(* IEC 61131-3 sources: Std_PalletMover/Class/RiwoParamAlarm, 1 file *)

(* ---- RiwoParamAlarm.st ---- *)
(*!
<Class
	Name               = "RiwoParamAlarm"
	Revision           = "0.2"
	RealtimeTask       = "false"
	CyclicTask         = "false"
	BackgroundTask     = "false"
	Sigmatek           = "false"
	OSInterface        = "false"
	HighPriority       = "false"
	Automatic          = "false"
	UpdateMode         = "Prescan"
	SharedCommandTable = "true"
	Objectsize         = "(450,660)">
	<Channels>
		<Server Name="GroupId" Visualized="true" Initialize="true" WriteProtected="false" Retentive="false"/>
		<Server Name="Id" Visualized="true" Initialize="false" WriteProtected="false" Retentive="false"/>
		<Server Name="Level" Visualized="true" Initialize="false" WriteProtected="false" Retentive="SRam"/>
		<Server Name="Parameter1" Visualized="false" Initialize="false" WriteProtected="false" Retentive="false"/>
		<Server Name="Parameter2" Visualized="false" Initialize="false" WriteProtected="false" Retentive="false"/>
		<Server Name="Parameter3" Visualized="false" Initialize="false" WriteProtected="false" Retentive="false"/>
		<Server Name="Parameter4" Visualized="false" Initialize="false" WriteProtected="false" Retentive="false"/>
		<Server Name="Report" Visualized="true" Initialize="false" WriteProtected="false" Retentive="SRam"/>
		<Server Name="ResetReq" Visualized="false" Initialize="true" WriteProtected="false" Retentive="false"/>
		<Client Name="_Group" Required="true" Internal="true"/>
		<Client Name="_Id" Required="true" Internal="true"/>
		<Client Name="objNextRiwoParamAlarm" Required="false" Internal="false"/>
		<Client Name="objRiwoEventLogger" Required="false" Internal="false"/>
	</Channels>
	<Dependencies>
		<Files>
			<File Path=".\Class\RiwoDefine\RiwoDef.h" Include="false"/>
		</Files>
	</Dependencies>
	<RevDoku>
		<Owner Company="Riwo Engineering B.V." Author="Stefan Veltmaat (SVE)"/>
		<Dokumentation Revision="0.1" Date="2018-07-27" Author="Stefan Veltmaat (SVE)" Company="Riwo Engineering B.V." Description="initial setup of parmeter error"/>
		<Dokumentation Date="2018-07-27" Author="Stefan Veltmaat (SVE)" Company="Riwo Engineering B.V."/>
	</RevDoku>
	<Network Name="RiwoParamAlarm">
		<!-- List of Components in this network -->
		<Components>
			<Object
				Name       = "_base"
				Class      = "_AlarmX3Para"
				Position   = "(534,120)"
				Visualized = "true"
				Remotely   = "true">
				<Channels>
					<Server Name="ClassSvr"/>
					<Client Name="Acknow"/>
					<Client Name="Config" Value="0"/>
					<Client Name="Group"/>
					<Client Name="Para1"/>
					<Client Name="Para2"/>
					<Client Name="Para3"/>
				</Channels>
			</Object>
			<Object
				Name       = "_Group"
				Class      = "Ram"
				Position   = "(390,690)"
				Visualized = "true"
				Remotely   = "true">
				<Channels>
					<Server Name="Data"/>
				</Channels>
			</Object>
			<Object
				Name       = "_Id"
				Class      = "Ram"
				Position   = "(390,480)"
				Visualized = "true"
				Remotely   = "true">
				<Channels>
					<Server Name="Data"/>
				</Channels>
			</Object>
		</Components>
		<Comments>
		</Comments>
		<!-- List of Connections in this network -->
		<Connections>
			<Connection Source="this.ClassSvr" Destination="_base.ClassSvr" Vertices="(1006,210),(834,210),"/>
			<Connection Source="this._Group" Destination="_Group.Data"/>
			<Connection Source="this.Id" Destination="_Id.Data" Vertices="(1006,270),(690,570),"/>
			<Connection Source="this.GroupId" Destination="_Group.Data" Vertices="(1006,330),(690,780),"/>
			<Connection Source="this._Id" Destination="_Id.Data"/>
		</Connections>
		<!-- Headerfiles -->
		<Options>
		</Options>
	</Network>
</Class>
*)
#pragma using _AlarmX3Para

RiwoParamAlarm : CLASS
: _AlarmX3Para
	TYPE
	  eAlarmLevel :  //! <Type Public="true" Name="eAlarmLevel"/>
	  (
	    eal_Error,
	    eal_Warning,
	    eal_Info
	  )$UDINT;
	  eAlarmReport :  //! <Type Public="true" Name="eAlarmReport"/>
	  (
	    ear_No,
	    ear_Yes
	  )$UDINT;
	END_TYPE
  //Servers:
	Id 	: SvrCh_DINT;
	GroupId 	: SvrCh_DINT;
	ResetReq 	: SvrCh_DINT;
	Level 	: SvrCh_eAlarmLevel_PTofCls_RiwoParamAlarm;
	Report 	: SvrCh_DINT;
	Parameter1 	: SvrCh_DINT;
	Parameter2 	: SvrCh_DINT;
	Parameter3 	: SvrCh_DINT;
	Parameter4 	: SvrCh_DINT;
  //Clients:
	objRiwoEventLogger 	: CltChCmd_RiwoEventLogger;
	objNextRiwoParamAlarm 	: CltChCmd_RiwoParamAlarm;
	_Id 	: CltChCmd_Ram;
	_Group 	: CltChCmd_Ram;
  //Variables:
  //Functions:

	FUNCTION VIRTUAL GLOBAL Init;

	FUNCTION VIRTUAL GLOBAL GetParaVal
		VAR_INPUT
			ppara 	: ^DINT;
		END_VAR
		VAR_OUTPUT
			retcode 	: UDINT;
		END_VAR;

	FUNCTION VIRTUAL GLOBAL QuitAlarm;

	FUNCTION _HandleAlarms
		VAR_INPUT
			newState 	: DINT;
		END_VAR;

	FUNCTION GLOBAL SetActive;

	FUNCTION GLOBAL SetInActive;

	FUNCTION GLOBAL SetActiveSingleParamAlarm
		VAR_INPUT
			inparam1 	: DINT;
		END_VAR;

	FUNCTION GLOBAL SetActiveTwoParamsAlarm
		VAR_INPUT
			inparam1 	: DINT;
			inparam2 	: DINT;
		END_VAR;

	FUNCTION GLOBAL SetActiveThreeParamsAlarm
		VAR_INPUT
			inparam1 	: DINT;
			inparam2 	: DINT;
			inparam3 	: DINT;
		END_VAR;

	FUNCTION GLOBAL GetActiveErrors
		VAR_INPUT
			objNr 	: UDINT;
		END_VAR
		VAR_OUTPUT
			errorsState 	: BDINT;
		END_VAR;

	FUNCTION GLOBAL GetActiveWarnings
		VAR_INPUT
			objNr 	: UDINT;
		END_VAR
		VAR_OUTPUT
			warningsState 	: BDINT;
		END_VAR;

	FUNCTION GLOBAL GetReportConfigs
		VAR_INPUT
			objNr 	: UDINT;
		END_VAR
		VAR_OUTPUT
			reportConfigs 	: BDINT;
		END_VAR;

	FUNCTION GLOBAL SetAlarmIds
		VAR_INPUT
			startId 	: DINT;
		END_VAR;

	FUNCTION VIRTUAL GLOBAL Id::Read
		VAR_OUTPUT
			output (EAX) 	: DINT;
		END_VAR;

	FUNCTION VIRTUAL GLOBAL Id::Write
		VAR_INPUT
			input (EAX) 	: DINT;
		END_VAR
		VAR_OUTPUT
			result (EAX) 	: DINT;
		END_VAR;

	FUNCTION VIRTUAL GLOBAL GroupId::Read
		VAR_OUTPUT
			output (EAX) 	: DINT;
		END_VAR;

	FUNCTION VIRTUAL GLOBAL GroupId::Write
		VAR_INPUT
			input (EAX) 	: DINT;
		END_VAR
		VAR_OUTPUT
			result (EAX) 	: DINT;
		END_VAR;

	FUNCTION VIRTUAL GLOBAL ResetReq::Read
		VAR_OUTPUT
			output (EAX) 	: DINT;
		END_VAR;

	FUNCTION VIRTUAL GLOBAL ResetReq::Write
		VAR_INPUT
			input (EAX) 	: DINT;
		END_VAR
		VAR_OUTPUT
			result (EAX) 	: DINT;
		END_VAR;
  //Tables:
	FUNCTION @STD
		VAR_OUTPUT
			ret_code	: CONFSTATES;
		END_VAR;
	FUNCTION GLOBAL TAB @CT_;
END_CLASS;

#pragma using Ram
#pragma usingLtd RiwoEventLogger

FUNCTION VIRTUAL GLOBAL RiwoParamAlarm::Init
  #if MAX_ALARMPARA >= 5
    #define ALARMPARA_NR_SUITABLE 1
  #endif

  #pragma warning(disable: 69);
  // compile error look into AlarmXBuffer.h and set MAX_ALARMPARA to 5
  if ALARMPARA_NR_SUITABLE then
    _AlarmX0Para::Init();
  end_if;
  #pragma warning(default: 69);

END_FUNCTION

FUNCTION GLOBAL RiwoParamAlarm::SetActive
  _HandleAlarms(1);
END_FUNCTION

FUNCTION GLOBAL RiwoParamAlarm::SetInActive
  _HandleAlarms(0);
END_FUNCTION

FUNCTION RiwoParamAlarm::_HandleAlarms
	VAR_INPUT
		newState 	: DINT;
	END_VAR

  if Level = eal_Warning & newState <> ClassSvr & newState = 1 then
    _RIWO_WARNING_MSG0("Alarm Id {0} activated", to_dint(Id));

    //write the new state to the ClassSvr so it is handled correct
    ClassSvr.Write(input:= newState);
  elsif Level = eal_Error  & newState <> ClassSvr & newState = 1 then
    _RIWO_ERROR_MSG0("Alarm Id {0} activated", to_dint(Id));

    //write the new state to the ClassSvr so it is handled correct
    ClassSvr.Write(input:= newState);
  elsif newState <> ClassSvr then
    _RIWO_INFO_MSG0("Alarm Id {0} de-activated", to_dint(Id));

    //write the new state to the ClassSvr so it is handled correct
    ClassSvr.Write(input:= newState);
  end_if;

  //all error updates must result in disabling the Reset request signal
  ResetReq := 0;

END_FUNCTION

FUNCTION VIRTUAL GLOBAL RiwoParamAlarm::GetParaVal
	VAR_INPUT
		ppara 	: ^DINT;
	END_VAR
	VAR_OUTPUT
		retcode 	: UDINT;
	END_VAR

  //Param position 0 contains level and report now, first 8 bits are Level, second 8 bits are report.
  ppara^ := Level$DINT AND 255;
  ppara^ := ppara^ OR Report$DINT SHL 8;

  //catch acces exception when sigmatek define is set back to its default of 3 instead of the needed 5
  //otherwise we are writing outside memory

  #if MAX_ALARMPARA >= 5
    ppara += 4;
    ppara^ := Parameter1;
    ppara += 4;
    ppara^ := Parameter2;
    ppara += 4;
    ppara^ := Parameter3;
    ppara += 4;
    ppara^ := Parameter4;
  #endif

  retcode := 5;
END_FUNCTION

FUNCTION GLOBAL RiwoParamAlarm::SetActiveSingleParamAlarm
	VAR_INPUT
		inparam1 	: DINT;
	END_VAR

   Parameter1  := inparam1;
   Parameter2  := -1;
   Parameter3  := -1;
   Parameter4  := -1;
   _HandleAlarms(1);
END_FUNCTION

FUNCTION GLOBAL RiwoParamAlarm::SetActiveTwoParamsAlarm
	VAR_INPUT
		inparam1 	: DINT;
		inparam2 	: DINT;
	END_VAR

   Parameter1  := inparam1;
   Parameter2  := inparam2;
   Parameter3  := -1;
   Parameter4  := -1;
   _HandleAlarms(1);
END_FUNCTION

FUNCTION GLOBAL RiwoParamAlarm::SetActiveThreeParamsAlarm
	VAR_INPUT
		inparam1 	: DINT;
		inparam2 	: DINT;
		inparam3 	: DINT;
	END_VAR

   Parameter1  := inparam1;
   Parameter2  := inparam2;
   Parameter3  := inparam3;
   Parameter4  := -1;
   _HandleAlarms(1);

END_FUNCTION

FUNCTION GLOBAL RiwoParamAlarm::GetActiveErrors
	VAR_INPUT
		objNr 	: UDINT;
	END_VAR
	VAR_OUTPUT
		errorsState 	: BDINT := 0;
	END_VAR

  if IsClientConnected(input:= #objNextRiwoParamAlarm) = true then
    errorsState := objNextRiwoParamAlarm.GetActiveErrors(objNr:= (objNr + 1));
  end_if;

  //set the coresponding error bit if the error is active
  if ClassSvr <> 0 & Level = eal_Error then
    errorsState := (errorsState or (1 shl objNr));
  end_if;

END_FUNCTION

FUNCTION GLOBAL RiwoParamAlarm::GetActiveWarnings
	VAR_INPUT
		objNr 	: UDINT;
	END_VAR
	VAR_OUTPUT
		warningsState 	: BDINT := 0;
	END_VAR

  if IsClientConnected(input:= #objNextRiwoParamAlarm) = true then
    warningsState := objNextRiwoParamAlarm.GetActiveWarnings(objNr:= (objNr + 1));
  end_if;

    //set the coresponding error bit if the error is active
  if ClassSvr <> 0 & Level = eal_Warning then
    warningsState := (warningsState or (1 shl objNr));
  end_if;

END_FUNCTION

FUNCTION GLOBAL RiwoParamAlarm::GetReportConfigs
	VAR_INPUT
		objNr 	: UDINT;
	END_VAR
	VAR_OUTPUT
		reportConfigs 	: BDINT := 0;
  END_VAR

  if IsClientConnected(input:= #objNextRiwoParamAlarm) = true then
    reportConfigs := objNextRiwoParamAlarm.GetReportConfigs(objNr:= (objNr + 1));
  end_if;

  //set the coresponding error bit if the error is active
  if Report <> 0 then
    reportConfigs := (reportConfigs or (1 shl objNr));
  end_if;

END_FUNCTION

//add aditional functionality to the QuitAlarm function
FUNCTION VIRTUAL GLOBAL RiwoParamAlarm::QuitAlarm
  _AlarmX0Para::QuitAlarm();
  if ClassSvr <> false then
    ResetReq.Write(input:= true);
  else
    ResetReq.Write(input:= false);
  end_if;
END_FUNCTION

FUNCTION GLOBAL RiwoParamAlarm::SetAlarmIds
	VAR_INPUT
		startId 	: DINT;
	END_VAR

  Id.Write(input:= startId);
  Config.Write(input:=startId);
  if IsClientConnected(input:= #objNextRiwoParamAlarm) = true then
    objNextRiwoParamAlarm.SetAlarmIds(startId:= (startId + 1));
  end_if;

END_FUNCTION

FUNCTION VIRTUAL GLOBAL RiwoParamAlarm::Id::Read
	VAR_OUTPUT
		output (EAX) 	: DINT;
	END_VAR

	output := Id;

END_FUNCTION

FUNCTION VIRTUAL GLOBAL RiwoParamAlarm::Id::Write
	VAR_INPUT
		input (EAX) 	: DINT;
	END_VAR
	VAR_OUTPUT
		result (EAX) 	: DINT;
	END_VAR

	Id := input;
	result := _Id.Data.Write(Id);

END_FUNCTION

FUNCTION VIRTUAL GLOBAL RiwoParamAlarm::GroupId::Read
	VAR_OUTPUT
		output (EAX) 	: DINT;
	END_VAR

	output := _Group.Data.Read();

END_FUNCTION

FUNCTION VIRTUAL GLOBAL RiwoParamAlarm::GroupId::Write
	VAR_INPUT
		input (EAX) 	: DINT;
	END_VAR
	VAR_OUTPUT
		result (EAX) 	: DINT;
	END_VAR

	GroupId := input;
	result := _Group.Data.Write(GroupId);

END_FUNCTION

FUNCTION VIRTUAL GLOBAL RiwoParamAlarm::ResetReq::Read
	VAR_OUTPUT
		output (EAX) 	: DINT;
	END_VAR

	output := ResetReq;

END_FUNCTION

FUNCTION VIRTUAL GLOBAL RiwoParamAlarm::ResetReq::Write
	VAR_INPUT
		input (EAX) 	: DINT;
	END_VAR
	VAR_OUTPUT
		result (EAX) 	: DINT;
	END_VAR

	ResetReq := input;
	result := ResetReq;

END_FUNCTION
